// Mitsubishi GX Works2 project: 0708-산술플러스   PLC: Q02/Q02H

PROGRAM MAIN
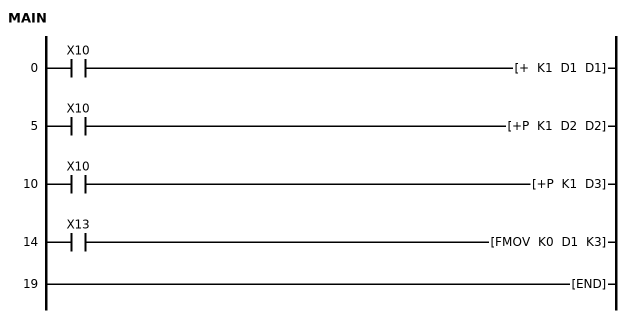
0     LD      X10
      +       K1 D1 D1
5     LD      X10
      +P      K1 D2 D2
10    LD      X10
      +P      K1 D3
14    LD      X13
      FMOV    K0 D1 K3
19    END
END_PROGRAM
